PROGRAM BurningProcess
VAR

END_VAR

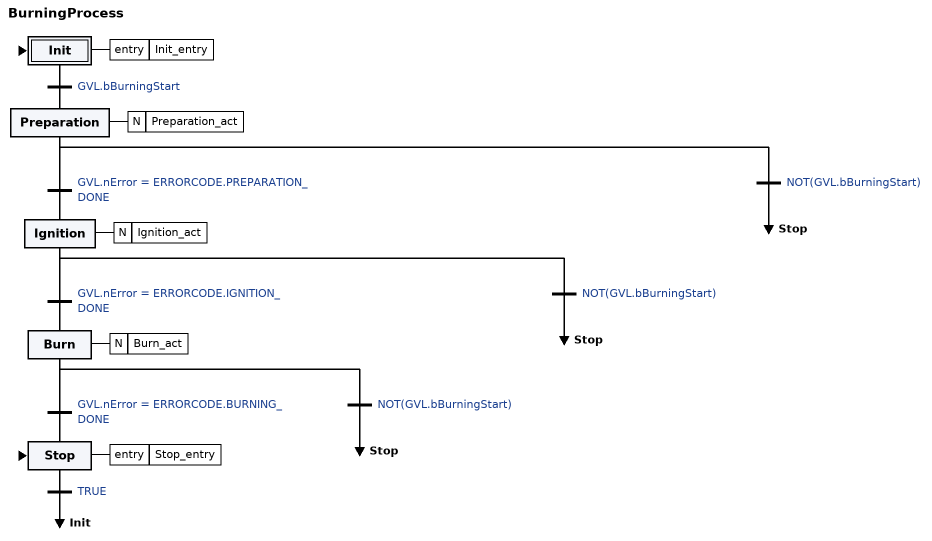
INITIAL_STEP Init:
    Init_entry(P1);  // entry action
END_STEP
TRANSITION FROM Init TO Preparation
    := GVL.bBurningStart;
END_TRANSITION
STEP Preparation:
    Preparation_act(N);
END_STEP
TRANSITION FROM Preparation TO Ignition
    := GVL.nError = ERRORCODE.PREPARATION_DONE;
END_TRANSITION
STEP Ignition:
    Ignition_act(N);
END_STEP
TRANSITION FROM Ignition TO Burn
    := GVL.nError = ERRORCODE.IGNITION_DONE;
END_TRANSITION
STEP Burn:
    Burn_act(N);
END_STEP
TRANSITION FROM Burn TO Stop
    := GVL.nError = ERRORCODE.BURNING_DONE;
END_TRANSITION
TRANSITION FROM Burn TO Stop
    := NOT(GVL.bBurningStart);
END_TRANSITION
TRANSITION FROM Ignition TO Stop
    := NOT(GVL.bBurningStart);
END_TRANSITION
TRANSITION FROM Preparation TO Stop
    := NOT(GVL.bBurningStart);
END_TRANSITION
STEP Stop:
    Stop_entry(P1);  // entry action
END_STEP
TRANSITION FROM Stop TO Init
    := TRUE;
END_TRANSITION

ACTION Burn_act:
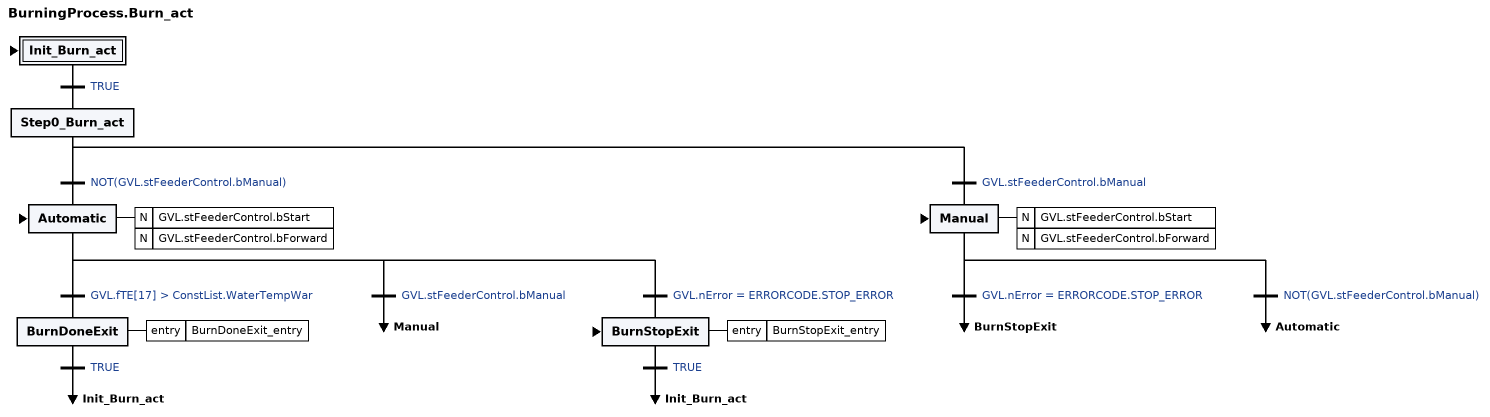
INITIAL_STEP Init_Burn_act:
END_STEP
TRANSITION FROM Init_Burn_act TO Step0_Burn_act
    := TRUE;
END_TRANSITION
STEP Step0_Burn_act:
END_STEP
TRANSITION FROM Step0_Burn_act TO Automatic
    := NOT(GVL.stFeederControl.bManual);
END_TRANSITION
STEP Automatic:
    GVL.stFeederControl.bStart(N);
    GVL.stFeederControl.bForward(N);
END_STEP
TRANSITION FROM Automatic TO BurnDoneExit
    := GVL.fTE[17] > ConstList.WaterTempWar;
END_TRANSITION
STEP BurnDoneExit:
    BurnDoneExit_entry(P1);  // entry action
END_STEP
TRANSITION FROM BurnDoneExit TO Init_Burn_act
    := TRUE;
END_TRANSITION
TRANSITION FROM Automatic TO Manual
    := GVL.stFeederControl.bManual;
END_TRANSITION
TRANSITION FROM Automatic TO BurnStopExit
    := GVL.nError = ERRORCODE.STOP_ERROR;
END_TRANSITION
STEP BurnStopExit:
    BurnStopExit_entry(P1);  // entry action
END_STEP
TRANSITION FROM BurnStopExit TO Init_Burn_act
    := TRUE;
END_TRANSITION
TRANSITION FROM Step0_Burn_act TO Manual
    := GVL.stFeederControl.bManual;
END_TRANSITION
STEP Manual:
    GVL.stFeederControl.bStart(N);
    GVL.stFeederControl.bForward(N);
END_STEP
TRANSITION FROM Manual TO BurnStopExit
    := GVL.nError = ERRORCODE.STOP_ERROR;
END_TRANSITION
TRANSITION FROM Manual TO Automatic
    := NOT(GVL.stFeederControl.bManual);
END_TRANSITION
// branch label Branch1_Burn_act
// branch label Branch2_Burn_act
// branch label Branch0_Burn_act
END_ACTION

ACTION BurnDoneExit_entry:
GVL.nError := ErRORCODE.BURNING_DONE;
END_ACTION

ACTION BurnStopExit_entry:
GVL.nError := errorcode.STOP_ERROR;
END_ACTION

ACTION ClearGases_active:
GVL.stPrimaryFan.nSpeed := 100;
GVL.stSecondaryFan.nSpeed := 100;
END_ACTION

ACTION FeederOn_exit:
GVL.nError := Errorcode.PREPARATION_DONE;
END_ACTION

ACTION FlameDetected_entry:
GVL.nError := ERRORCODE.PREPARATION_FLAME;
END_ACTION

ACTION Ignite_exit:
GVL.nError := ERRORCODE.IGNITION_DONE;
END_ACTION

ACTION Ignition_act:
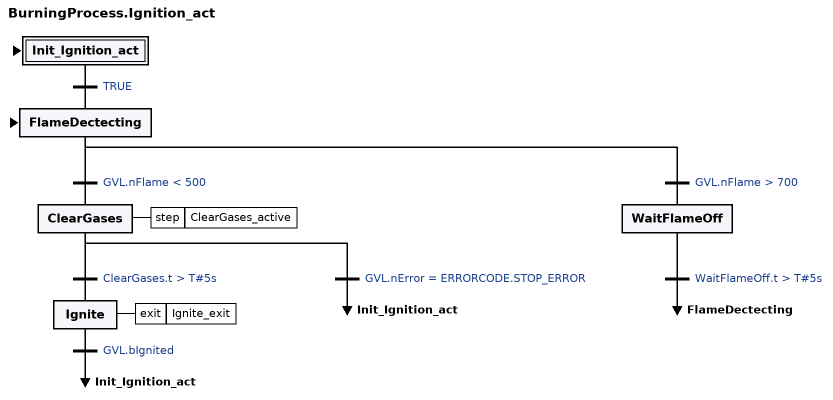
INITIAL_STEP Init_Ignition_act:
END_STEP
TRANSITION FROM Init_Ignition_act TO FlameDectecting
    := TRUE;
END_TRANSITION
STEP FlameDectecting:
END_STEP
TRANSITION FROM FlameDectecting TO ClearGases
    := GVL.nFlame < 500;
END_TRANSITION
STEP ClearGases:
    ClearGases_active(N);  // step action
END_STEP
TRANSITION FROM ClearGases TO Ignite
    := ClearGases.t > T#5s;
END_TRANSITION
STEP Ignite:
    Ignite_exit(P0);  // exit action
END_STEP
TRANSITION FROM Ignite TO Init_Ignition_act
    := GVL.bIgnited;
END_TRANSITION
TRANSITION FROM ClearGases TO Init_Ignition_act
    := GVL.nError = ERRORCODE.STOP_ERROR;
END_TRANSITION
TRANSITION FROM FlameDectecting TO WaitFlameOff
    := GVL.nFlame > 700;
END_TRANSITION
STEP WaitFlameOff:
END_STEP
TRANSITION FROM WaitFlameOff TO FlameDectecting
    := WaitFlameOff.t > T#5s;
END_TRANSITION
// branch label Branch1_Ignition_act
// branch label Branch0_Ignition_act
END_ACTION

ACTION Init_entry:
GVL.stPrimaryFan.nSpeed := 0;
GVL.stSecondaryFan.nSpeed := 0;
GVL.stFeederControl.bStart := FALSE;
GVL.stFeederControl.bForward := FALSE;
GVL.nError := 0;
END_ACTION

ACTION Preparation_act:
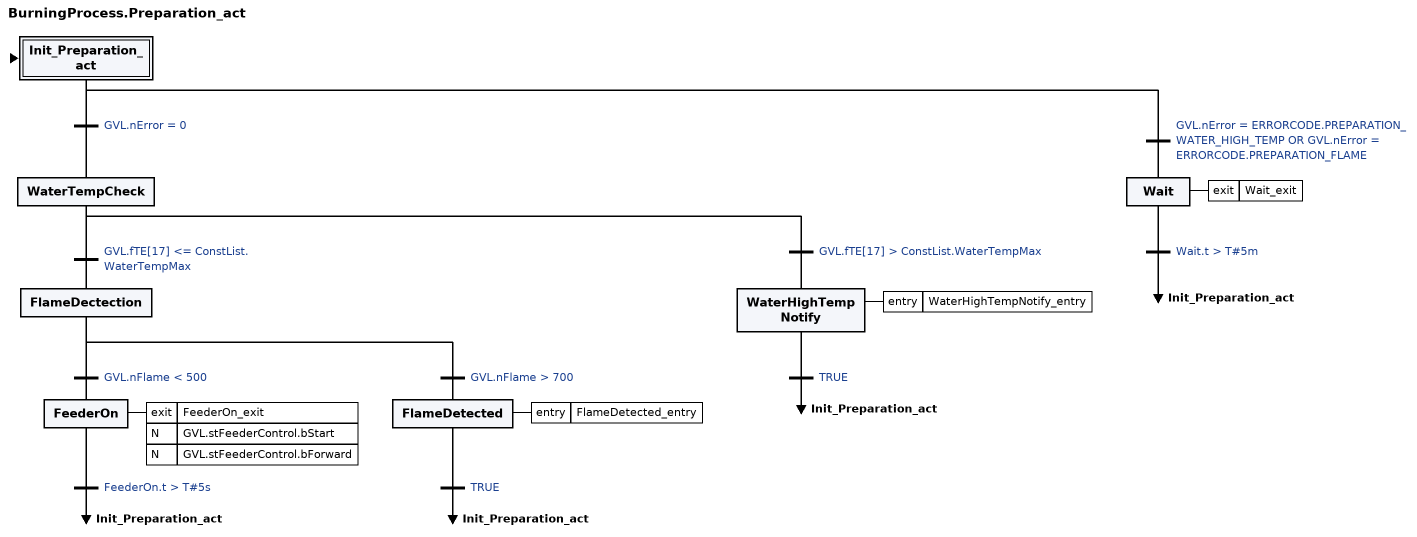
INITIAL_STEP Init_Preparation_act:
END_STEP
TRANSITION FROM Init_Preparation_act TO WaterTempCheck
    := GVL.nError = 0;
END_TRANSITION
TRANSITION FROM Init_Preparation_act TO Wait
    := GVL.nError = ERRORCODE.PREPARATION_WATER_HIGH_TEMP OR GVL.nError = ERRORCODE.PREPARATION_FLAME;
END_TRANSITION
STEP Wait:
    Wait_exit(P0);  // exit action
END_STEP
TRANSITION FROM Wait TO Init_Preparation_act
    := Wait.t > T#5m;
END_TRANSITION
STEP WaterTempCheck:
END_STEP
TRANSITION FROM WaterTempCheck TO FlameDectection
    := GVL.fTE[17] <= ConstList.WaterTempMax;
END_TRANSITION
STEP FlameDectection:
END_STEP
TRANSITION FROM FlameDectection TO FeederOn
    := GVL.nFlame < 500;
END_TRANSITION
STEP FeederOn:
    FeederOn_exit(P0);  // exit action
    GVL.stFeederControl.bStart(N);
    GVL.stFeederControl.bForward(N);
END_STEP
TRANSITION FROM FeederOn TO Init_Preparation_act
    := FeederOn.t > T#5s;
END_TRANSITION
TRANSITION FROM FlameDectection TO FlameDetected
    := GVL.nFlame > 700;
END_TRANSITION
STEP FlameDetected:
    FlameDetected_entry(P1);  // entry action
END_STEP
TRANSITION FROM FlameDetected TO Init_Preparation_act
    := TRUE;
END_TRANSITION
TRANSITION FROM WaterTempCheck TO WaterHighTempNotify
    := GVL.fTE[17] > ConstList.WaterTempMax;
END_TRANSITION
STEP WaterHighTempNotify:
    WaterHighTempNotify_entry(P1);  // entry action
END_STEP
TRANSITION FROM WaterHighTempNotify TO Init_Preparation_act
    := TRUE;
END_TRANSITION
// branch label Branch2_Preparation_act
// branch label Branch1_Preparation_act
// branch label Branch0_Preparation_act
END_ACTION

ACTION Stop_entry:
GVL.stPrimaryFan.nSpeed := 0;
GVL.stSecondaryFan.nSpeed := 0;
GVL.stFeederControl.bStart := FALSE;
GVL.stFeederControl.bForward := FALSE;
GVL.nError := 0;
//GVL.bP1 := FALSE;
//GVL.bP2 := FALSE;
END_ACTION

ACTION Wait_exit:
GVL.nError := ERRORCODE.SUCCESS;
END_ACTION

ACTION WaterHighTempNotify_entry:
GVL.nError := ERRorcode.PREPARATION_WATER_HIGH_TEMP;
END_ACTION

END_PROGRAM

(* stored: Version 1.1.0.1, ProductVersion 3.1.4022.18
   POU BurningProcess: Id {df4b61a4-5b36-4a6a-ae54-2fd3ee2ec963}, SpecialFunc None
   Folder Burn: Id {84a12832-f015-4bbd-bdb3-f8929ca16218}
   Folder Ignition: Id {96868aad-5924-4e9b-aa4a-3c0174adb574}
   Folder Preparation: Id {972d84d4-53cf-4abf-b6f4-1f67d8de76f6}
   Folder Stop: Id {10acaca8-9e71-4bca-8b2c-535364191c06}
   Action Burn_act: Id {63db8a19-2463-448a-82e6-a3523950f777}
   Action BurnDoneExit_entry: Id {8ba174d2-0adf-4969-8c35-7f58247cda41}
   Action BurnStopExit_entry: Id {33c10884-72c6-4f8b-9032-0985dfec2fae}
   Action ClearGases_active: Id {682d4a56-a14f-4ef7-ba57-26c57c77baa2}
   Action FeederOn_exit: Id {90473c85-096e-4adb-881b-a1761b46a9e4}
   Action FlameDetected_entry: Id {b3c5e8b6-dcca-4fcb-a20e-56359283b0e8}
   Action Ignite_exit: Id {6170c120-07a6-4ab9-8e8a-742c3f0ff17f}
   Action Ignition_act: Id {5245fdce-9b79-4325-a9d9-aedcc6a6c96e}
   Action Init_entry: Id {bea47634-cb86-4f7b-ab4e-d27486bd4887}
   Action Preparation_act: Id {e2f09129-ce75-438c-be94-669687c53dec}
   Action Stop_entry: Id {e64abd77-5200-462c-a458-51bc7bffbd9c}
   Action Wait_exit: Id {6fefab59-aea3-4a87-a021-c87938eabda7}
   Action WaterHighTempNotify_entry: Id {f2240639-9222-45bf-8a05-9a9629abb13f} *)
